PROGRAM MAIN
VAR
	
    heartbeat : BYTE;
	
	// Outputs.
	one AT %Q* : BOOL;
	two AT %Q* : BOOL;
	three AT %Q* : BOOL;
	four AT %Q* : BOOL;
	
	prox AT %I* : BOOL;  // Input
	
	// Dynamic Throttle
	Throttle AT %I* : INT;
	LastThrottle : INT;
	
	AxisB : AXIS_REF;

	McPower : MC_Power;
	McReset : MC_Reset;
	McJogging : MC_Jog;
	McVelocity : MC_MoveVelocity;
	McStop : MC_Stop;
	McHome : MC_Home;

	
    CurrentVelocityCmd : DINT;

	iState : DINT; // My State

	McMoveAbs : MC_MoveAbsolute;
	McMoveRel : MC_MoveRelative;
	iNumMoves : DINT:= 5;
	iCurrMove : DINT;
	fMoveDistEachTime : REAL:= 10;
	fRelMoveDist : REAL;
	
	TcJoy : FB_TcJoy;

END_VAR

heartbeat := heartbeat + 1;

CurrentVelocityCmd := MAP(Throttle,29800,22600,0,2800);
IF CurrentVelocityCmd < 50 THEN
	CurrentVelocityCmd := 0;
END_IF

AxisB.ReadStatus();

McPower(Axis:=AxisB,Enable:=TRUE,Enable_Positive:=TRUE,Enable_Negative:=TRUE);
McReset(Axis:=AxisB);
McJogging(Axis:=AxisB);
McHome(Axis:=AxisB,bCalibrationCam := prox);

McMoveAbs(Axis:=AxisB);
McMoveRel(Axis:=AxisB);

TcJoy();

CASE iState OF
	
    0:  // Initial

		iState := 10;

    10:  // Start Drive Reset

		McHome(Axis:=AxisB,Execute:=FALSE);
		McReset(Axis:=AxisB,Execute:=TRUE);
		IF McReset.Done THEN
			iState :=20;
		ELSIF McReset.Error THEN
			iState := 999;
		END_IF

    20:  // Wait for Drive to Reset

		IF McPower.Status AND (CurrentVelocityCmd > 1000 OR TcJoy.Y_Button) THEN
			iState := 100;
		END_IF	
		
    30:  // Wait for drive JOG command.
    
		IF TcJoy.iRightTrigger_Axis > 0 THEN
	
			IF TcJoy.iRightStick_X_Axis > 0 THEN
				McJogging.JogForward := TRUE;
				McJogging.Velocity := ABS(MAP(TcJoy.iRightStick_X_Axis,6000,32767,0,720));
			ELSE
				McJogging.JogForward := FALSE;
			END_IF
			IF TcJoy.iRightStick_X_Axis < 0 THEN
				McJogging.JogBackwards := TRUE;
				McJogging.Velocity := ABS(MAP(TcJoy.iRightStick_X_Axis,-6000,-32767,0,720));				
			ELSE
				McJogging.JogBackwards := FALSE;
			END_IF
			IF TcJoy.iRightStick_X_Axis = 0 THEN
				McJogging.JogForward := FALSE;
				McJogging.JogBackwards := FALSE;
			END_IF
			
			McJogging.Mode := MC_JOGMODE_CONTINOUS;
			McJogging.Acceleration := 500;
			McJogging.Deceleration := 500;
			McJogging.Jerk := 1000000;
			McJogging(Axis:=AxisB);
			
		ELSE
			McJogging.JogForward := FALSE;
			McJogging.JogBackwards := FALSE;
			iState := 200;
		END_IF 
		
	40:  // Wait for velocity command.
	
	//	McVelocity(Axis:=AxisB,
	//			Velocity:=CurrentVelocityCmd,
	///			Acceleration:=10000,
	//			Deceleration:=10000,
	//			Jerk:=1000000,
	//			Direction:=MC_Direction.MC_Positive_Direction,
	//			Execute:=prox AND (LastThrottle<>Throttle));
	//	IF NOT prox THEN
	//		McVelocity(Axis:=AxisB,Execute:=FALSE);
	//		iState := 900;
	//	END_IF				
	//	
		
		IF TcJoy.iLeftTrigger_Axis > 0 THEN
			
			McStop(Axis:=AxisB,Execute:=FALSE);
			
			IF TcJoy.iRightStick_X_Axis > 0 THEN
				McVelocity.Velocity := ABS(MAP(TcJoy.iRightStick_X_Axis,6000,32767,0,720));
			END_IF
			IF TcJoy.iRightStick_X_Axis < 0 THEN
				McVelocity.Velocity := ABS(MAP(TcJoy.iRightStick_X_Axis,-6000,-32767,0,720));				
			END_IF
			IF TcJoy.iRightStick_X_Axis = 0 THEN
				McVelocity.Velocity := 0;
			END_IF

			McVelocity(Axis:=AxisB, Execute:=LastThrottle<>Throttle);
			
		ELSE
			McVelocity(Axis:=AxisB, Execute:=FALSE);
			McStop(Axis:=AxisB,Execute:=TRUE);
			iState := 200;
		END_IF 
		
		LastThrottle:=Throttle;
		
	100:  // Start Homing Process.
		
		McHome(Axis:=AxisB,bCalibrationCam:=prox,Execute:=TRUE);
		IF McHome.Busy THEN
			iState := 110;
		END_IF
		
	110: // Homing running, wait for homing to complete.
	
		IF McHome.Done AND NOT McHome.Error THEN
			McHome(Axis:=AxisB,Execute:=FALSE);
			iState := 200;
		ELSIF McHome.Error THEN
			McHome(Axis:=AxisB,Execute:=FALSE);
			iState := 999;
		END_IF
		
	200: // Homing Complete.  Ready to Run.
		
		IF TcJoy.Y_Button THEN // Home
			iState := 100;	
		END_IF
		IF TcJoy.B_Button THEN // Run dance move
			iState := 300;
		END_IF
		IF TcJoy.iRightTrigger_Axis > 0 THEN // Jog with joystick
			iState := 30;
		END_IF
		IF TcJoy.iLeftTrigger_Axis > 0 THEN // ABS with joystick
			iState := 600;
		END_IF
		
 	300:  // Start ABS Move to center to prep for processing part
	
	    McMoveAbs(Axis:=AxisB,
					Position := 100,
					Velocity := 100,
					Acceleration := 500,
					Deceleration := 500,
					Jerk := 100000,
					Execute:=TRUE);
					
		iState := 310;
		
	310:  // Wait for abs move to complete.
	
	    IF McMoveAbs.Done AND NOT McMoveAbs.Error THEN
			McMoveAbs(Axis:=AxisB,Execute:=FALSE);
			iCurrMove := 1;
			iState := 400;
		ELSIF McMoveAbs.Error THEN
			McMoveAbs(Axis:=AxisB,Execute:=FALSE);
			iState := 999;	
		END_IF
		
	400:  // Start Rel Moves.
	
	    // More to do?
		IF iCurrMove < iNumMoves THEN
			// increment move counter for next time.
			iCurrMove := iCurrMove + 1;
			// Calculate Distance
			fRelMoveDist := DINT_TO_REAL(iCurrMove) * fMoveDistEachTime;
			iState := 410;
		ELSE
			// Nothing to do.
			iState := 500;
		END_IF
		
	410:  // Start rel move in pos direction
		
	    McMoveRel(Axis:=AxisB,
					Distance := fRelMoveDist,
					Velocity := 720,
					Acceleration := 2000,
					Deceleration := 2000,
					Jerk := 1000000,
					Execute:=TRUE);
					
		iState := 420;
		
	420:  // Wait on rel move to complete
	
		IF McMoveRel.Done AND NOT McMoveRel.Error THEN
			McMoveRel(Axis:=AxisB,Execute:=FALSE);
			iState := 450;
		ELSIF McMoveRel.Error THEN
			McMoveRel(Axis:=AxisB,Execute:=FALSE);
			iState := 999;	
		END_IF
		
	450:  // Move negative rel back to start position
					
		McMoveRel(Axis:=AxisB,
					Distance := -fRelMoveDist,
					Velocity := 720,
					Acceleration := 2000,
					Deceleration := 2000,
					Jerk := 1000000,
					Execute:=TRUE);
					
		iState := 460;
		
	460:  // Wait on rel move to complete
	
		IF McMoveRel.Done AND NOT McMoveRel.Error THEN
			McMoveRel(Axis:=AxisB,Execute:=FALSE);
			iState := 400;
		ELSIF McMoveRel.Error THEN
			McMoveRel(Axis:=AxisB,Execute:=FALSE);
			iState := 999;	
		END_IF

	500:  // Start ABS Move Back to home
	
	    McMoveAbs(Axis:=AxisB,
					Position := 0,
					Velocity := 100,
					Acceleration := 100,
					Deceleration := 100,
					Jerk := 100000,
					Execute:=TRUE);
					
		iState := 510;
		
	510:  // Wait for abs move to complete.
	
	    IF McMoveAbs.Done AND NOT McMoveAbs.Error THEN
			McMoveAbs(Axis:=AxisB,Execute:=FALSE);
			iCurrMove := 1;
			iState := 200;
		ELSIF McMoveAbs.Error THEN
			McMoveAbs(Axis:=AxisB,Execute:=FALSE);
			iState := 999;	
		END_IF		
		
		
	600:   // Start ABS Move from joystick
	
		IF TcJoy.iLeftTrigger_Axis > 0 THEN
	
			IF TcJoy.iRightStick_X_Axis > 0 THEN
				McMoveAbs.Position := ABS(MAP(TcJoy.iRightStick_X_Axis,6000,32767,100,200));
			END_IF
			IF TcJoy.iRightStick_X_Axis < 0 THEN
				McMoveAbs.Position := ABS(MAP(TcJoy.iRightStick_X_Axis,-32767,-6000,0,100));				
			END_IF
			IF TcJoy.iRightStick_X_Axis = 0 THEN
				McMoveAbs.Position := 100;
			END_IF

			McMoveAbs(Axis:=AxisB,
					Velocity := 500,
					Acceleration := 500,
					Deceleration := 2000,
					Jerk := 1000000,
					Execute:=TRUE);
					
			iState := 610;
			
		ELSE
			McMoveAbs(Axis:=AxisB,Execute:=FALSE);
			iState := 200;
		END_IF 
	

		
	610:  // Wait for abs move to complete.
	
	    IF McMoveAbs.Done AND NOT McMoveAbs.Error THEN
			McMoveAbs(Axis:=AxisB,Execute:=FALSE);
			iState := 600;
		ELSIF McMoveAbs.Error THEN
			McMoveAbs(Axis:=AxisB,Execute:=FALSE);
			iState := 999;	
		END_IF	
	
	900:  // Stop servo.
	
	    McStop(Axis:=AxisB,Execute:=TRUE);
		IF prox THEN
			McStop(Axis:=AxisB,Execute:=FALSE);
			iState := 40;
		END_IF
	
	999: // Handle Error (TODO)

END_CASE

END_PROGRAM

(* stored: Version 1.1.0.1, ProductVersion 3.1.4022.9
   POU MAIN: Id {53de4ad1-482e-4350-a93f-8d5c37cbb918}, SpecialFunc None *)
